// TIA Portal V15.1 export
// export: Created 2020-06-12T07:35:55.4130859Z, ExportSetting None, DisplayName Totally Integrated Automation Portal, DisplayVersion V15.1, DisplayName TIA Portal Openness, DisplayVersion V15.1, DisplayName STEP 7 Professional, DisplayVersion V15.1, DisplayName STEP 7 Safety, DisplayVersion V15.1, DisplayName WinCC Advanced, DisplayVersion V15.1
FUNCTION "SLAG_ctrl" : Void   // FC120, FBD
TITLE = Slag addition base control
{ S7_Optimized_Access := 'TRUE' }
// stored: SetENOAutomatically False
   VAR_TEMP
      tReqFeedOn : Bool;
      tReqFeedOff : Bool;
      tReqPush : Bool;
      tReqDummy : Bool;
      tReqFloodOn : Bool;
      tReqFloodOff : Bool;
      tReqMan : Bool;
      tReqAuto : Bool;
      tReqSetTara : Bool;
      tReqCondMode : Bool;
      tReqDirectMode : Bool;
      tReqRateFree : Bool;
      tReqRateFixed : Bool;
      tStage : Word;
      tDeskActive : Bool;
      tDeskFeedOn : Bool;
      tDeskPush : Bool;
      tManCmdOn : Bool;
      tManCmdOff : Bool;
      tLock : Bool;
      tCmdOn : Bool;
      tCmdOff : Bool;
      tReqOn : Bool;
      tReqOff : Bool;
      tCondStop : Bool;
      tTargetWeightReached : Bool;
      tLoadedWeight : Real;
      tLoadStarting : Bool;
      tLoadStopping : Bool;
      tReqReset : Bool;
      tLock2 : Bool;
      tReqFixSpd2 : Bool;
      tReqFixSpd1 : Bool;
      tInvalidWeight : Bool;
      tNoisedWgt : Real;
      tNoise : Real;
      tDeskChangeSpd : Bool;
      tDeskSelSpd2 : Bool;
      tPwrOk : Bool;
      tDeskSelSpd1 : Bool;
      tDeskFloodOn : Bool;
      tDeskFloodOff : Bool;
      tRestWeight : Real;
      tFeederIsStopped : Bool;
      tBinISEmpty : Bool;
      tHammerBitFast : Bool;
      tHammerBitSlow : Bool;
      tBeat : Bool;
      tLoadRate : Real;
      tReqFloodOff_ : Bool;
   END_VAR
   VAR_TEMP   // added for the SCL form of the ladder/FBD networks
      _w1 : Bool;
      _w2 : Bool;
   END_VAR
BEGIN

REGION Network 1: Common fault
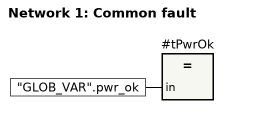
   #tPwrOk := "GLOB_VAR".pwr_ok;
END_REGION

REGION Network 2: HMI request treat
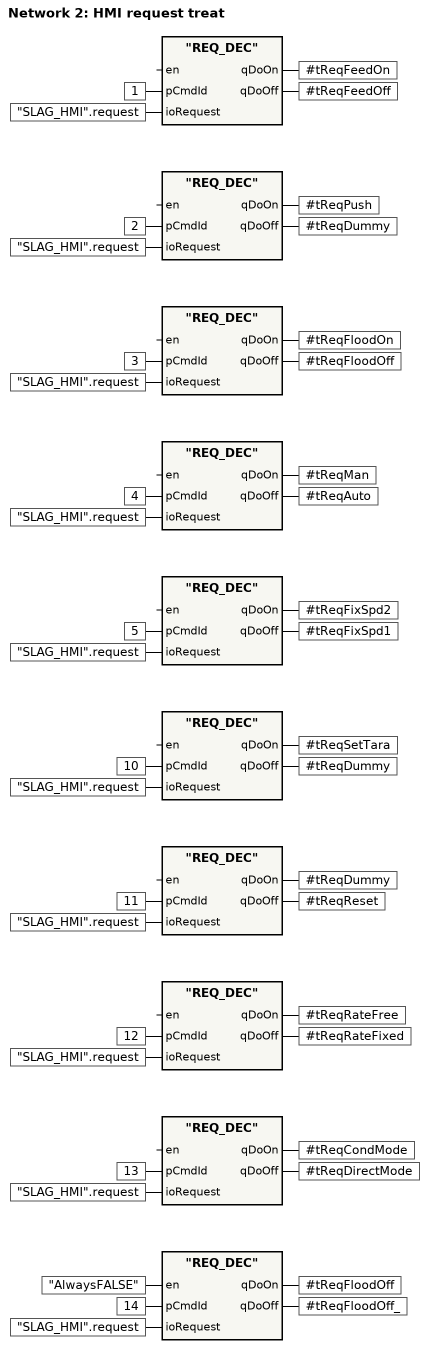
   "REQ_DEC"(pCmdId := 1, ioRequest := "SLAG_HMI".request, qDoOn => #tReqFeedOn, qDoOff => #tReqFeedOff);
   "REQ_DEC"(pCmdId := 2, ioRequest := "SLAG_HMI".request, qDoOn => #tReqPush, qDoOff => #tReqDummy);
   "REQ_DEC"(pCmdId := 3, ioRequest := "SLAG_HMI".request, qDoOn => #tReqFloodOn, qDoOff => #tReqFloodOff);
   "REQ_DEC"(pCmdId := 4, ioRequest := "SLAG_HMI".request, qDoOn => #tReqMan, qDoOff => #tReqAuto);
   "REQ_DEC"(pCmdId := 5, ioRequest := "SLAG_HMI".request, qDoOn => #tReqFixSpd2, qDoOff => #tReqFixSpd1);
   "REQ_DEC"(pCmdId := 10, ioRequest := "SLAG_HMI".request, qDoOn => #tReqSetTara, qDoOff => #tReqDummy);
   "REQ_DEC"(pCmdId := 11, ioRequest := "SLAG_HMI".request, qDoOn => #tReqDummy, qDoOff => #tReqReset);
   "REQ_DEC"(pCmdId := 12, ioRequest := "SLAG_HMI".request, qDoOn => #tReqRateFree, qDoOff => #tReqRateFixed);
   "REQ_DEC"(pCmdId := 13, ioRequest := "SLAG_HMI".request, qDoOn => #tReqCondMode, qDoOff => #tReqDirectMode);
   IF "AlwaysFALSE" THEN
       "REQ_DEC"(pCmdId := 14, ioRequest := "SLAG_HMI".request, qDoOn => #tReqFloodOff, qDoOff => #tReqFloodOff_);
   END_IF;
END_REGION

REGION Network 3: An operators desks are active
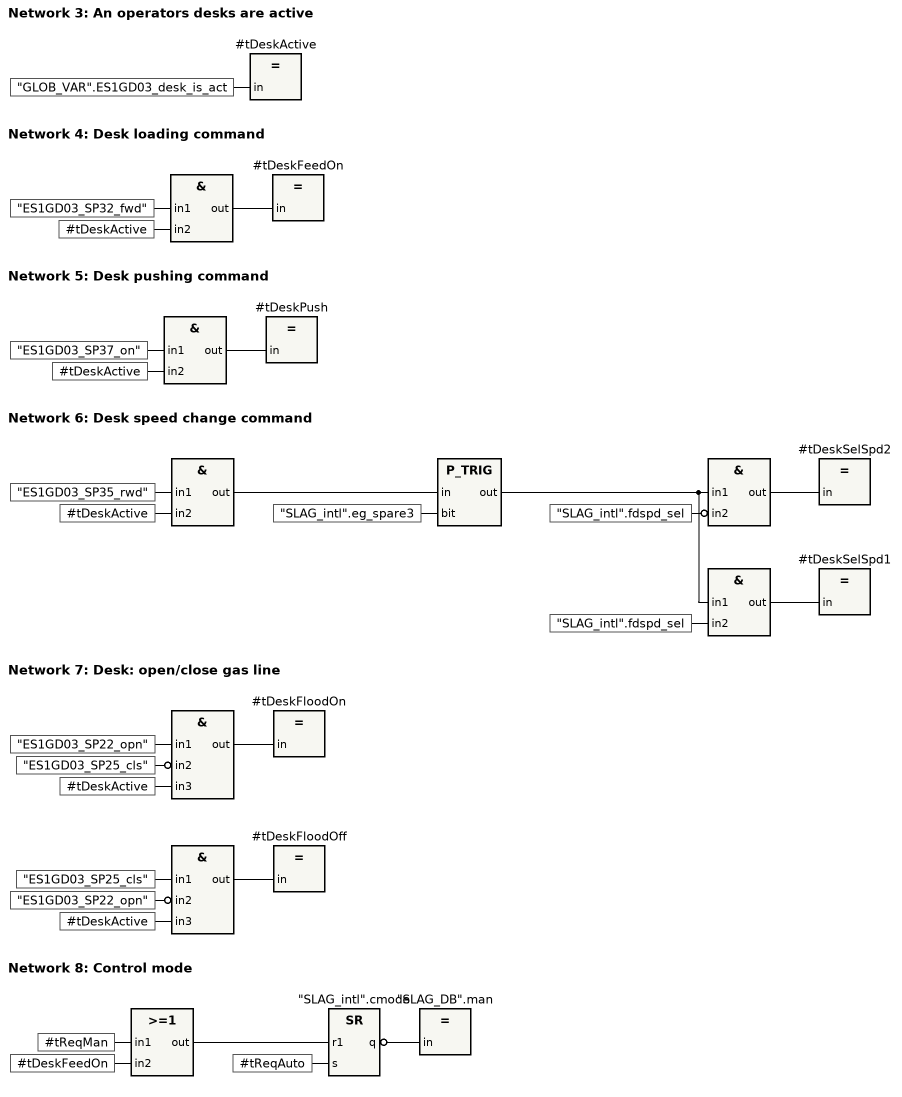
   #tDeskActive := "GLOB_VAR".ES1GD03_desk_is_act;
END_REGION

REGION Network 4: Desk loading command
   #tDeskFeedOn := "ES1GD03_SP32_fwd" AND #tDeskActive;
END_REGION

REGION Network 5: Desk pushing command
   // The sense of this command for a vibro-feeder is not so clear...
   // 
   // But we can use this button to activate the pusher.
   #tDeskPush := "ES1GD03_SP37_on" AND #tDeskActive;
END_REGION

REGION Network 6: Desk speed change command
   #_w1 := "ES1GD03_SP35_rwd" AND #tDeskActive;
   #_w2 := #_w1 AND NOT "SLAG_intl".eg_spare3;   // rising edge
   "SLAG_intl".eg_spare3 := #_w1;
   #tDeskSelSpd2 := #_w2 AND NOT "SLAG_intl".fdspd_sel;
   #tDeskSelSpd1 := #_w2 AND "SLAG_intl".fdspd_sel;
END_REGION

REGION Network 7: Desk: open/close gas line
   #tDeskFloodOn := "ES1GD03_SP22_opn" AND NOT "ES1GD03_SP25_cls" AND #tDeskActive;
   #tDeskFloodOff := "ES1GD03_SP25_cls" AND NOT "ES1GD03_SP22_opn" AND #tDeskActive;
END_REGION

REGION Network 8: Control mode
   // "SLAG_intl".cmode
   IF #tReqAuto THEN
       "SLAG_intl".cmode := TRUE;   // SR flip-flop
   END_IF;
   IF #tReqMan OR #tDeskFeedOn THEN "SLAG_intl".cmode := FALSE; END_IF;
   "SLAG_DB".man := NOT "SLAG_intl".cmode;
END_REGION

REGION Network 9: Loading mode
   // For an external program the conditional loading is always using
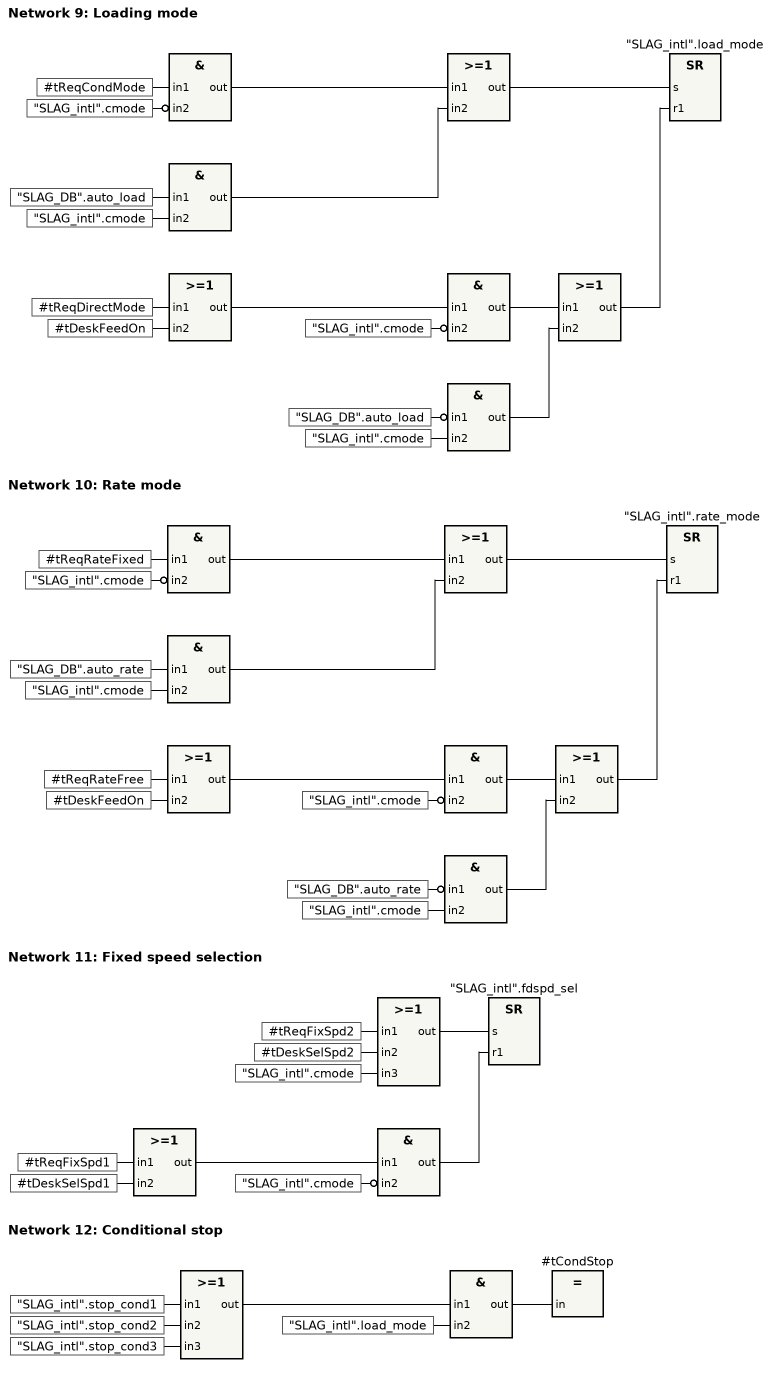
   IF (#tReqCondMode AND NOT "SLAG_intl".cmode) OR ("SLAG_DB".auto_load AND "SLAG_intl".cmode) THEN
       "SLAG_intl".load_mode := TRUE;   // SR flip-flop
   END_IF;
   IF ((#tReqDirectMode OR #tDeskFeedOn) AND NOT "SLAG_intl".cmode) OR (NOT "SLAG_DB".auto_load AND "SLAG_intl".cmode) THEN
       "SLAG_intl".load_mode := FALSE;
   END_IF;
END_REGION

REGION Network 10: Rate mode
   IF (#tReqRateFixed AND NOT "SLAG_intl".cmode) OR ("SLAG_DB".auto_rate AND "SLAG_intl".cmode) THEN
       "SLAG_intl".rate_mode := TRUE;   // SR flip-flop
   END_IF;
   IF ((#tReqRateFree OR #tDeskFeedOn) AND NOT "SLAG_intl".cmode) OR (NOT "SLAG_DB".auto_rate AND "SLAG_intl".cmode) THEN
       "SLAG_intl".rate_mode := FALSE;
   END_IF;
END_REGION

REGION Network 11: Fixed speed selection
   IF #tReqFixSpd2 OR #tDeskSelSpd2 OR "SLAG_intl".cmode THEN
       "SLAG_intl".fdspd_sel := TRUE;   // SR flip-flop
   END_IF;
   IF (#tReqFixSpd1 OR #tDeskSelSpd1) AND NOT "SLAG_intl".cmode THEN "SLAG_intl".fdspd_sel := FALSE; END_IF;
END_REGION

REGION Network 12: Conditional stop
   // NB: This network here becuase of optimization
   #tCondStop := ("SLAG_intl".stop_cond1 OR "SLAG_intl".stop_cond2 OR "SLAG_intl".stop_cond3) AND "SLAG_intl".load_mode;
END_REGION

REGION Network 13: Lock by invalid measurement
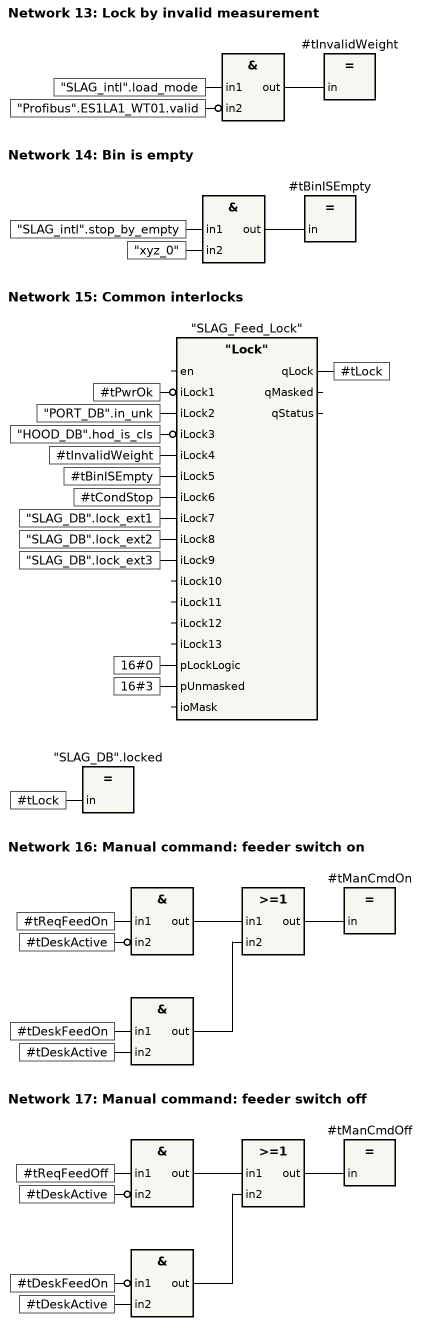
   #tInvalidWeight := "SLAG_intl".load_mode AND NOT "Profibus".ES1LA1_WT01.valid;
END_REGION

REGION Network 14: Bin is empty
   #tBinISEmpty := "SLAG_intl".stop_by_empty AND "xyz_0";
END_REGION

REGION Network 15: Common interlocks
   "SLAG_Feed_Lock"(iLock1 := NOT #tPwrOk,   // "Lock"
                    iLock2 := "PORT_DB".in_unk,
                    iLock3 := NOT "HOOD_DB".hod_is_cls,
                    iLock4 := #tInvalidWeight,
                    iLock5 := #tBinISEmpty,
                    iLock6 := #tCondStop,
                    iLock7 := "SLAG_DB".lock_ext1,
                    iLock8 := "SLAG_DB".lock_ext2,
                    iLock9 := "SLAG_DB".lock_ext3,
                    pLockLogic := 16#0,
                    pUnmasked := 16#3,
                    qLock => #tLock);
   "SLAG_DB".locked := #tLock;
END_REGION

REGION Network 16: Manual command: feeder switch on
   #tManCmdOn := (#tReqFeedOn AND NOT #tDeskActive) OR (#tDeskFeedOn AND #tDeskActive);
END_REGION

REGION Network 17: Manual command: feeder switch off
   #tManCmdOff := (#tReqFeedOff AND NOT #tDeskActive) OR (NOT #tDeskFeedOn AND #tDeskActive);
END_REGION

REGION Network 18: Manual start/stop
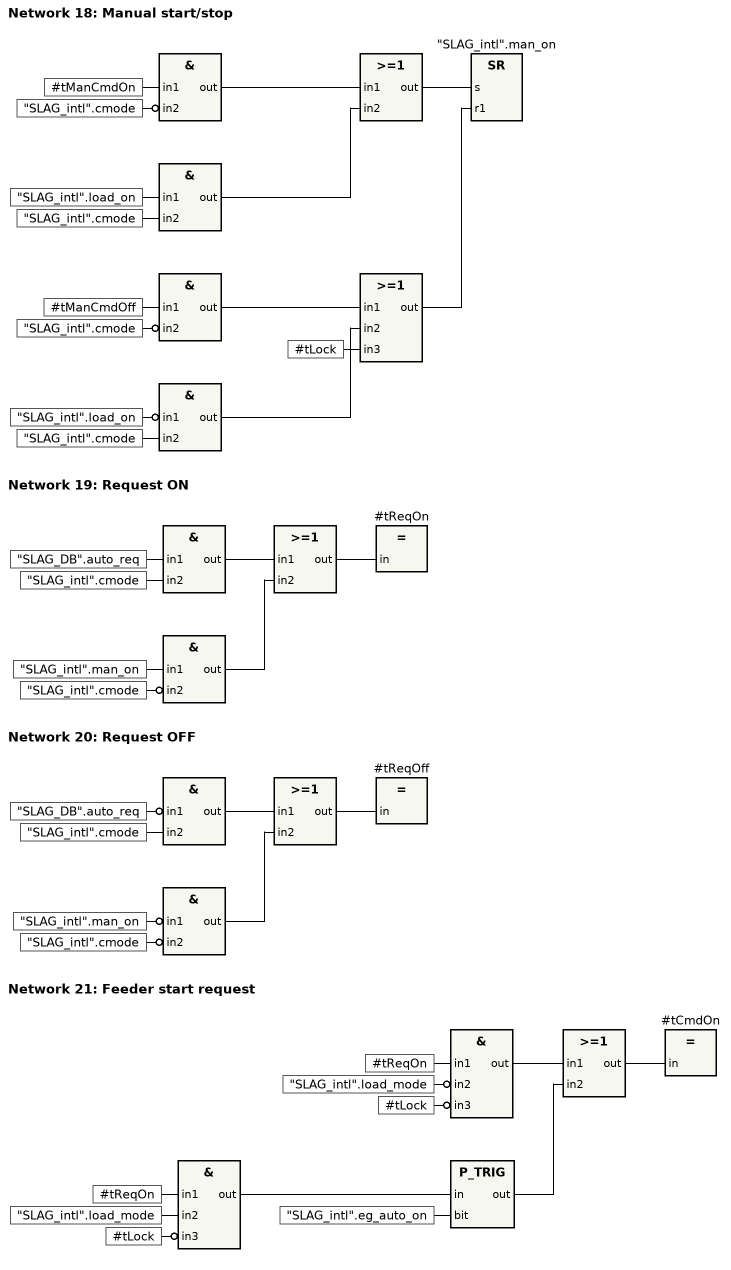
   IF (#tManCmdOn AND NOT "SLAG_intl".cmode) OR ("SLAG_intl".load_on AND "SLAG_intl".cmode) THEN
       "SLAG_intl".man_on := TRUE;   // SR flip-flop
   END_IF;
   IF (#tManCmdOff AND NOT "SLAG_intl".cmode) OR (NOT "SLAG_intl".load_on AND "SLAG_intl".cmode) OR #tLock THEN
       "SLAG_intl".man_on := FALSE;
   END_IF;
END_REGION

REGION Network 19: Request ON
   #tReqOn := ("SLAG_DB".auto_req AND "SLAG_intl".cmode) OR ("SLAG_intl".man_on AND NOT "SLAG_intl".cmode);
END_REGION

REGION Network 20: Request OFF
   #tReqOff := (NOT "SLAG_DB".auto_req AND "SLAG_intl".cmode) OR (NOT "SLAG_intl".man_on AND NOT "SLAG_intl".cmode);
END_REGION

REGION Network 21: Feeder start request
   // I use tLock because want to implmement a restartable program
   #_w1 := #tReqOn AND "SLAG_intl".load_mode AND NOT #tLock;
   #_w2 := #_w1 AND NOT "SLAG_intl".eg_auto_on;   // rising edge
   "SLAG_intl".eg_auto_on := #_w1;
   #tCmdOn := (#tReqOn AND NOT "SLAG_intl".load_mode AND NOT #tLock) OR #_w2;
END_REGION

REGION Network 22: Feeder stop request
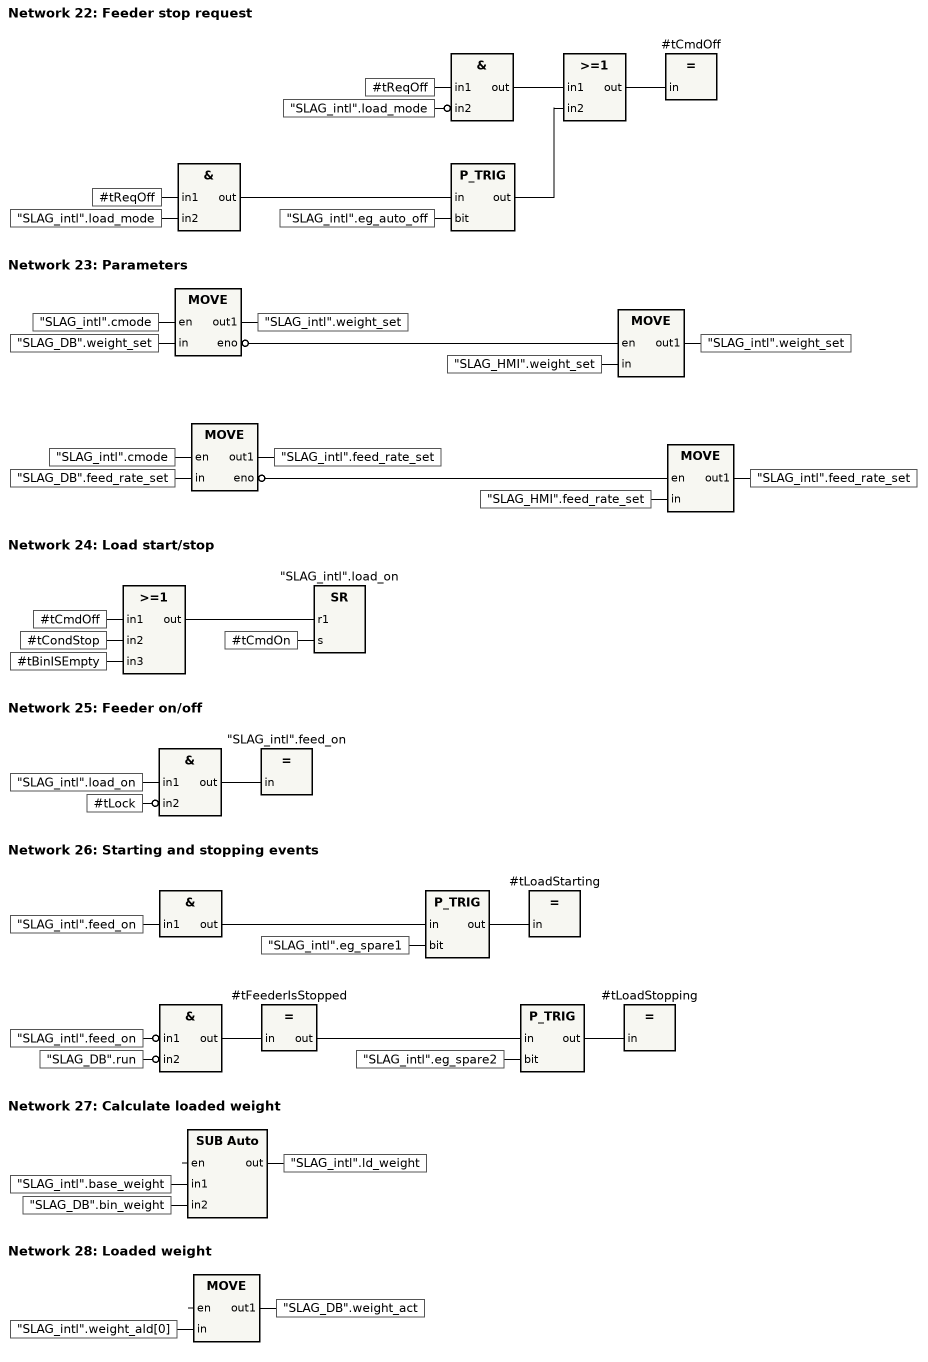
   #_w1 := #tReqOff AND "SLAG_intl".load_mode;
   #_w2 := #_w1 AND NOT "SLAG_intl".eg_auto_off;   // rising edge
   "SLAG_intl".eg_auto_off := #_w1;
   #tCmdOff := (#tReqOff AND NOT "SLAG_intl".load_mode) OR #_w2;
END_REGION

REGION Network 23: Parameters
   IF "SLAG_intl".cmode THEN "SLAG_intl".weight_set := "SLAG_DB".weight_set; END_IF;
   IF NOT "SLAG_intl".cmode THEN "SLAG_intl".weight_set := "SLAG_HMI".weight_set; END_IF;
   IF "SLAG_intl".cmode THEN "SLAG_intl".feed_rate_set := "SLAG_DB".feed_rate_set; END_IF;
   IF NOT "SLAG_intl".cmode THEN "SLAG_intl".feed_rate_set := "SLAG_HMI".feed_rate_set; END_IF;
END_REGION

REGION Network 24: Load start/stop
   IF #tCmdOn THEN
       "SLAG_intl".load_on := TRUE;   // SR flip-flop
   END_IF;
   IF #tCmdOff OR #tCondStop OR #tBinISEmpty THEN "SLAG_intl".load_on := FALSE; END_IF;
END_REGION

REGION Network 25: Feeder on/off
   "SLAG_intl".feed_on := "SLAG_intl".load_on AND NOT #tLock;
END_REGION

REGION Network 26: Starting and stopping events
   #_w1 := "SLAG_intl".feed_on AND NOT "SLAG_intl".eg_spare1;   // rising edge
   "SLAG_intl".eg_spare1 := "SLAG_intl".feed_on;
   #tLoadStarting := #_w1;
   #tFeederIsStopped := NOT "SLAG_intl".feed_on AND NOT "SLAG_DB".run;
   #_w2 := #tFeederIsStopped AND NOT "SLAG_intl".eg_spare2;   // rising edge
   "SLAG_intl".eg_spare2 := #tFeederIsStopped;
   #tLoadStopping := #_w2;
END_REGION

REGION Network 27: Calculate loaded weight
   "SLAG_intl".ld_weight := "SLAG_intl".base_weight - "SLAG_DB".bin_weight;
END_REGION

REGION Network 28: Loaded weight
   "SLAG_DB".weight_act := "SLAG_intl".weight_ald[0];
END_REGION

REGION Network 29: Calculate accumulating loaded weight
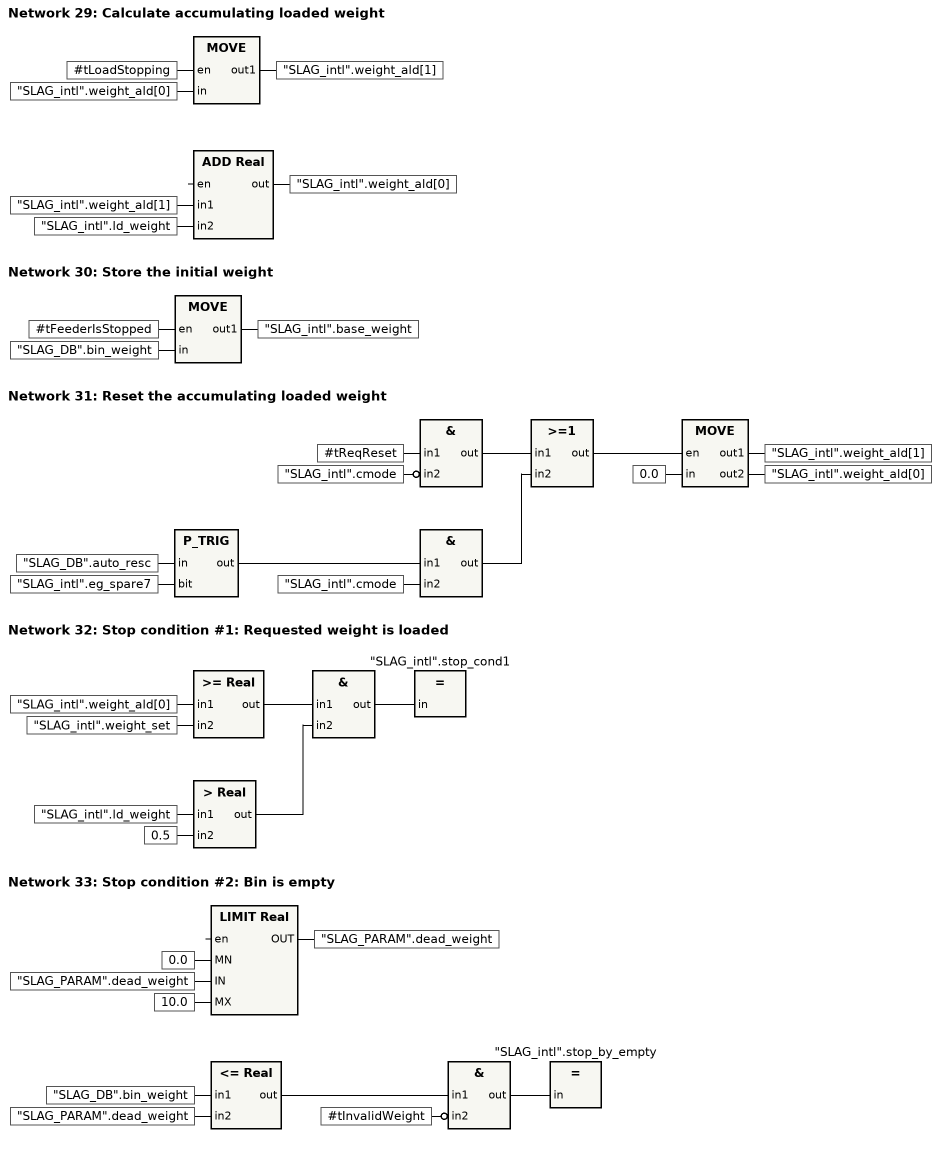
   IF #tLoadStopping THEN "SLAG_intl".weight_ald[1] := "SLAG_intl".weight_ald[0]; END_IF;
   "SLAG_intl".weight_ald[0] := "SLAG_intl".weight_ald[1] + "SLAG_intl".ld_weight;
END_REGION

REGION Network 30: Store the initial weight
   // The #tLoadStarting has been replace by {NOT "SLAG_intl".feed_on }
   IF #tFeederIsStopped THEN "SLAG_intl".base_weight := "SLAG_DB".bin_weight; END_IF;
END_REGION

REGION Network 31: Reset the accumulating loaded weight
   #_w1 := "SLAG_DB".auto_resc AND NOT "SLAG_intl".eg_spare7;   // rising edge
   "SLAG_intl".eg_spare7 := "SLAG_DB".auto_resc;
   IF (#tReqReset AND NOT "SLAG_intl".cmode) OR (#_w1 AND "SLAG_intl".cmode) THEN
       "SLAG_intl".weight_ald[1] := 0.0;
       "SLAG_intl".weight_ald[0] := 0.0;
   END_IF;
END_REGION

REGION Network 32: Stop condition #1: Requested weight is loaded
   "SLAG_intl".stop_cond1 := ("SLAG_intl".weight_ald[0] >= "SLAG_intl".weight_set) AND ("SLAG_intl".ld_weight > 0.5);
END_REGION

REGION Network 33: Stop condition #2: Bin is empty
   "SLAG_PARAM".dead_weight := LIMIT(MN := 0.0, IN := "SLAG_PARAM".dead_weight, MX := 10.0);
   "SLAG_intl".stop_by_empty := ("SLAG_DB".bin_weight <= "SLAG_PARAM".dead_weight) AND NOT #tInvalidWeight;
END_REGION

REGION Network 34: Detect a prestop weight
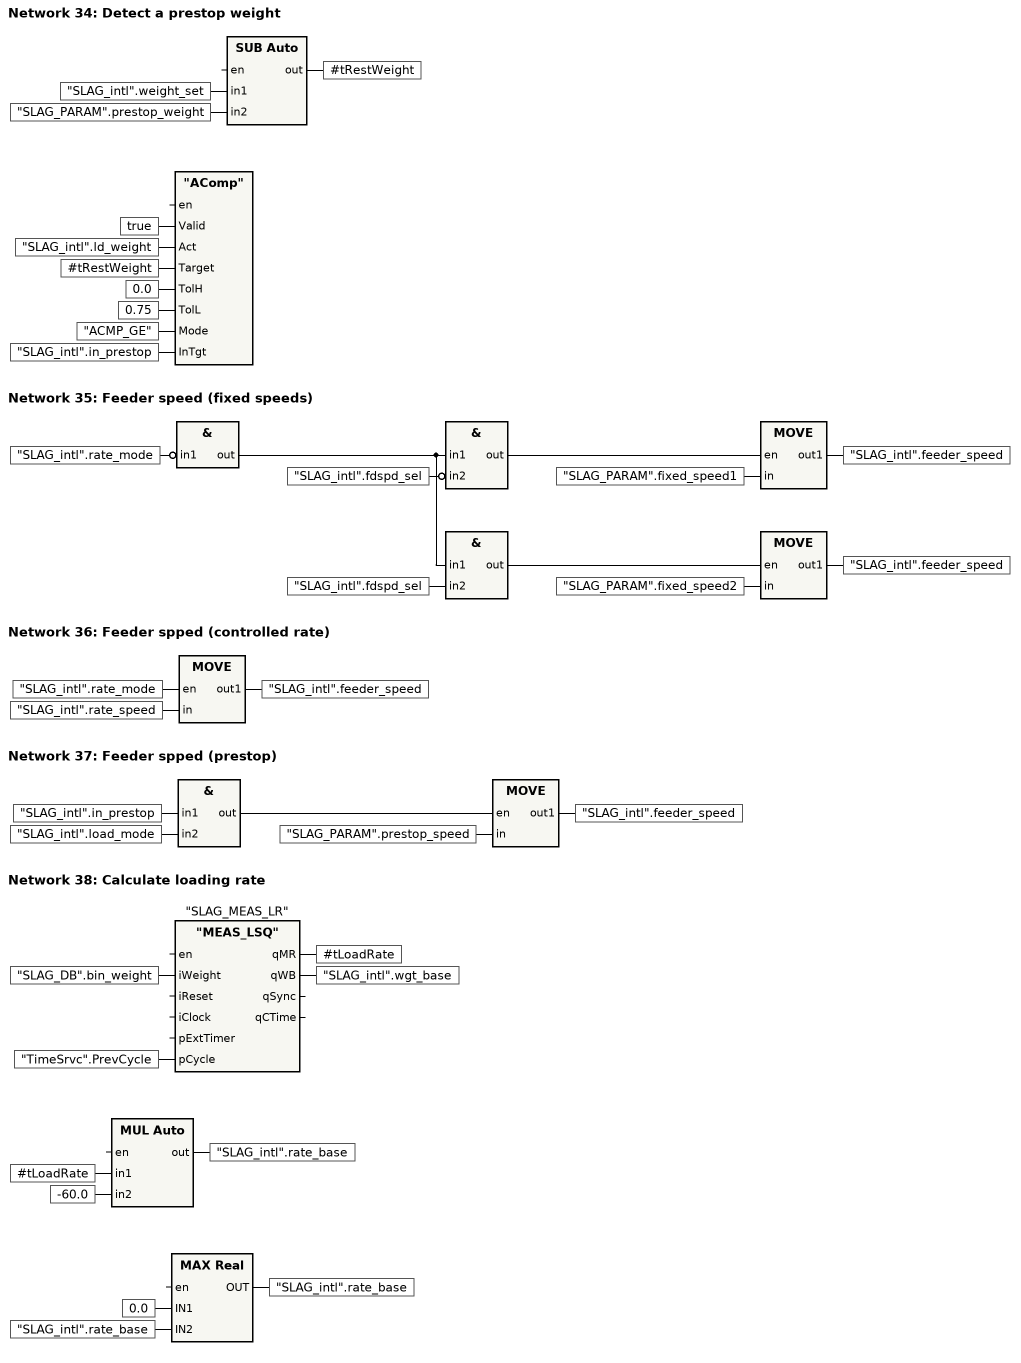
   #tRestWeight := "SLAG_intl".weight_set - "SLAG_PARAM".prestop_weight;
   "AComp"(Valid := true,
           Act := "SLAG_intl".ld_weight,
           Target := #tRestWeight,
           TolH := 0.0,
           TolL := 0.75,
           Mode := "ACMP_GE",
           InTgt := "SLAG_intl".in_prestop);
END_REGION

REGION Network 35: Feeder speed (fixed speeds)
   #_w1 := NOT "SLAG_intl".rate_mode;
   IF #_w1 AND NOT "SLAG_intl".fdspd_sel THEN "SLAG_intl".feeder_speed := "SLAG_PARAM".fixed_speed1; END_IF;
   IF #_w1 AND "SLAG_intl".fdspd_sel THEN "SLAG_intl".feeder_speed := "SLAG_PARAM".fixed_speed2; END_IF;
END_REGION

REGION Network 36: Feeder spped (controlled rate)
   IF "SLAG_intl".rate_mode THEN "SLAG_intl".feeder_speed := "SLAG_intl".rate_speed; END_IF;
END_REGION

REGION Network 37: Feeder spped (prestop)
   IF "SLAG_intl".in_prestop AND "SLAG_intl".load_mode THEN
       "SLAG_intl".feeder_speed := "SLAG_PARAM".prestop_speed;
   END_IF;
END_REGION

REGION Network 38: Calculate loading rate
   "SLAG_MEAS_LR"(iWeight := "SLAG_DB".bin_weight,   // "MEAS_LSQ"
                  pCycle := "TimeSrvc".PrevCycle,
                  qMR => #tLoadRate,
                  qWB => "SLAG_intl".wgt_base);
   "SLAG_intl".rate_base := #tLoadRate * (-60.0);
   "SLAG_intl".rate_base := MAX(IN1 := 0.0, IN2 := "SLAG_intl".rate_base);
END_REGION

REGION Network 39: Stacking detection
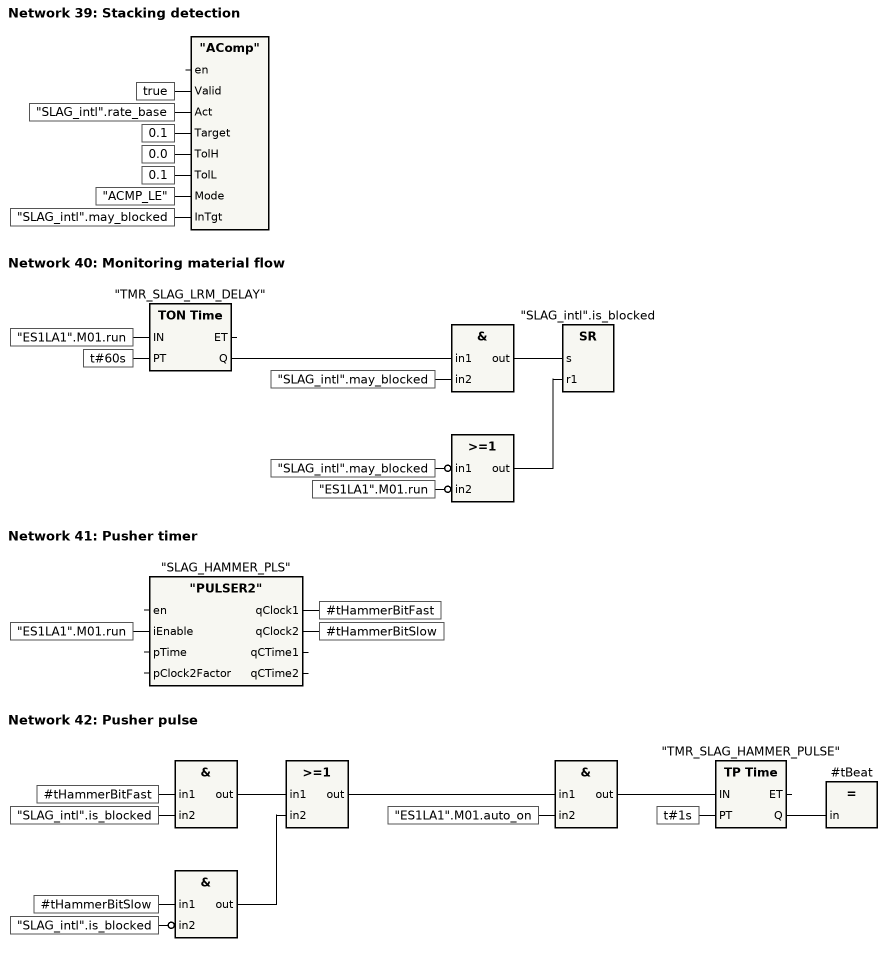
   "AComp"(Valid := true,
           Act := "SLAG_intl".rate_base,
           Target := 0.1,
           TolH := 0.0,
           TolL := 0.1,
           Mode := "ACMP_LE",
           InTgt := "SLAG_intl".may_blocked);
END_REGION

REGION Network 40: Monitoring material flow
   "TMR_SLAG_LRM_DELAY".TON(IN := "ES1LA1".M01.run, PT := t#60s);
   IF "TMR_SLAG_LRM_DELAY".Q AND "SLAG_intl".may_blocked THEN
       "SLAG_intl".is_blocked := TRUE;   // SR flip-flop
   END_IF;
   IF NOT "SLAG_intl".may_blocked OR NOT "ES1LA1".M01.run THEN "SLAG_intl".is_blocked := FALSE; END_IF;
END_REGION

REGION Network 41: Pusher timer
   "SLAG_HAMMER_PLS"(iEnable := "ES1LA1".M01.run, qClock1 => #tHammerBitFast, qClock2 => #tHammerBitSlow);   // "PULSER2"
END_REGION

REGION Network 42: Pusher pulse
   "TMR_SLAG_HAMMER_PULSE".TP(IN := ((#tHammerBitFast AND "SLAG_intl".is_blocked) OR (#tHammerBitSlow AND NOT "SLAG_intl".is_blocked)) AND "ES1LA1".M01.auto_on,
                           PT := t#1s);
   #tBeat := "TMR_SLAG_HAMMER_PULSE".Q;
END_REGION

REGION Network 43: Gas flooding
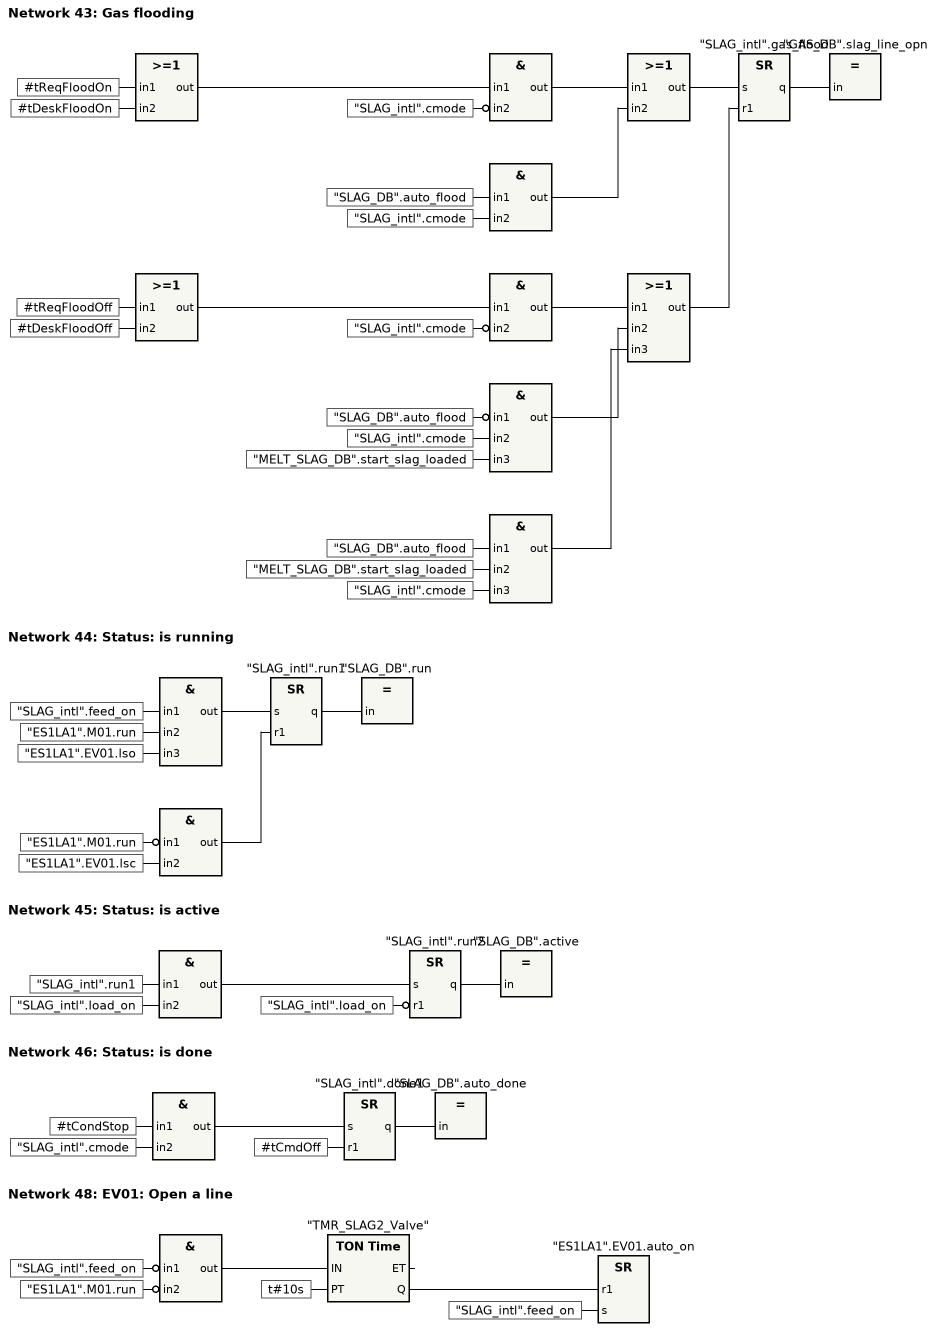
   IF ((#tReqFloodOn OR #tDeskFloodOn) AND NOT "SLAG_intl".cmode) OR ("SLAG_DB".auto_flood AND "SLAG_intl".cmode) THEN
       "SLAG_intl".gas_flood := TRUE;   // SR flip-flop
   END_IF;
   IF ((#tReqFloodOff OR #tDeskFloodOff) AND NOT "SLAG_intl".cmode) OR (NOT "SLAG_DB".auto_flood AND "SLAG_intl".cmode AND "MELT_SLAG_DB".start_slag_loaded) OR ("SLAG_DB".auto_flood AND "MELT_SLAG_DB".start_slag_loaded AND "SLAG_intl".cmode) THEN
       "SLAG_intl".gas_flood := FALSE;
   END_IF;
   "GAS_DB".slag_line_opn := "SLAG_intl".gas_flood;
END_REGION

REGION Network 44: Status: is running
   IF "SLAG_intl".feed_on AND "ES1LA1".M01.run AND "ES1LA1".EV01.lso THEN
       "SLAG_intl".run1 := TRUE;   // SR flip-flop
   END_IF;
   IF NOT "ES1LA1".M01.run AND "ES1LA1".EV01.lsc THEN "SLAG_intl".run1 := FALSE; END_IF;
   "SLAG_DB".run := "SLAG_intl".run1;
END_REGION

REGION Network 45: Status: is active
   IF "SLAG_intl".run1 AND "SLAG_intl".load_on THEN
       "SLAG_intl".run2 := TRUE;   // SR flip-flop
   END_IF;
   IF NOT "SLAG_intl".load_on THEN "SLAG_intl".run2 := FALSE; END_IF;
   "SLAG_DB".active := "SLAG_intl".run2;
END_REGION

REGION Network 46: Status: is done
   IF #tCondStop AND "SLAG_intl".cmode THEN
       "SLAG_intl".done1 := TRUE;   // SR flip-flop
   END_IF;
   IF #tCmdOff THEN "SLAG_intl".done1 := FALSE; END_IF;
   "SLAG_DB".auto_done := "SLAG_intl".done1;
END_REGION

REGION Network 47: [ DEVICES control]
END_REGION

REGION Network 48: EV01: Open a line
   "TMR_SLAG2_Valve".TON(IN := NOT "SLAG_intl".feed_on AND NOT "ES1LA1".M01.run, PT := t#10s);
   IF "SLAG_intl".feed_on THEN
       "ES1LA1".EV01.auto_on := TRUE;   // SR flip-flop
   END_IF;
   IF "TMR_SLAG2_Valve".Q THEN "ES1LA1".EV01.auto_on := FALSE; END_IF;
END_REGION

REGION Network 49: EV01: lock open
   // I do not want to use the lock, to avoid a valve closing while a loading
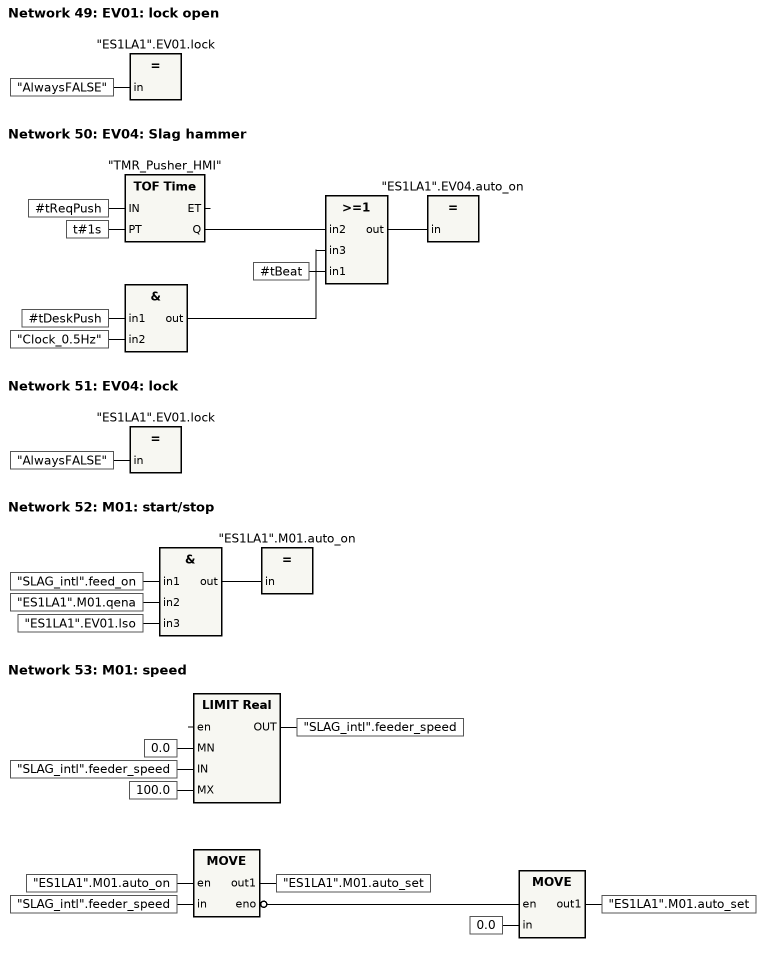
   "ES1LA1".EV01.lock := "AlwaysFALSE";
END_REGION

REGION Network 50: EV04: Slag hammer
   "TMR_Pusher_HMI".TOF(IN := #tReqPush, PT := t#1s);
   "ES1LA1".EV04.auto_on := "TMR_Pusher_HMI".Q OR (#tDeskPush AND "Clock_0.5Hz") OR #tBeat;
END_REGION

REGION Network 51: EV04: lock
   // there are not the restrictions
   "ES1LA1".EV01.lock := "AlwaysFALSE";
END_REGION

REGION Network 52: M01: start/stop
   "ES1LA1".M01.auto_on := "SLAG_intl".feed_on AND "ES1LA1".M01.qena AND "ES1LA1".EV01.lso;
END_REGION

REGION Network 53: M01: speed
   "SLAG_intl".feeder_speed := LIMIT(MN := 0.0, IN := "SLAG_intl".feeder_speed, MX := 100.0);
   IF "ES1LA1".M01.auto_on THEN "ES1LA1".M01.auto_set := "SLAG_intl".feeder_speed; END_IF;
   IF NOT "ES1LA1".M01.auto_on THEN "ES1LA1".M01.auto_set := 0.0; END_IF;
END_REGION

REGION Network 54: M01: lock forward
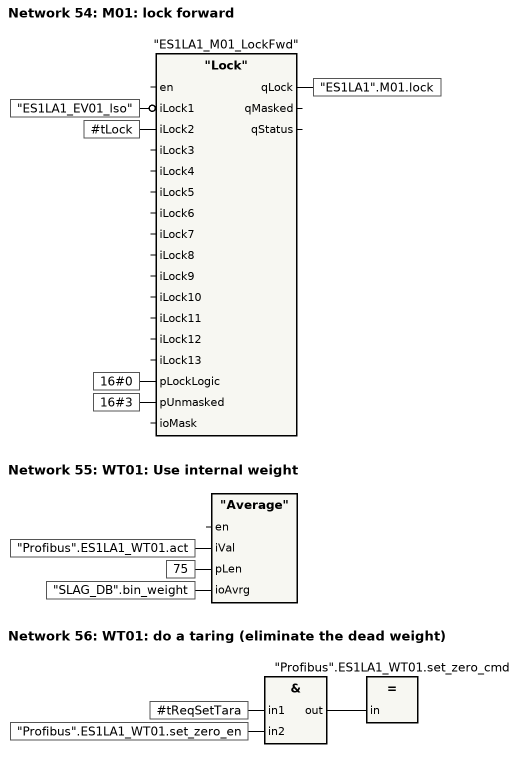
   "ES1LA1_M01_LockFwd"(iLock1 := NOT "ES1LA1_EV01_lso",   // "Lock"
                        iLock2 := #tLock,
                        pLockLogic := 16#0,
                        pUnmasked := 16#3,
                        qLock => "ES1LA1".M01.lock);
END_REGION

REGION Network 55: WT01: Use internal weight
   "Average"(iVal := "Profibus".ES1LA1_WT01.act, pLen := 75, ioAvrg := "SLAG_DB".bin_weight);
END_REGION

REGION Network 56: WT01: do a taring (eliminate the dead weight)
   "Profibus".ES1LA1_WT01.set_zero_cmd := #tReqSetTara AND "Profibus".ES1LA1_WT01.set_zero_en;
END_REGION

REGION Network 57: HMI: status
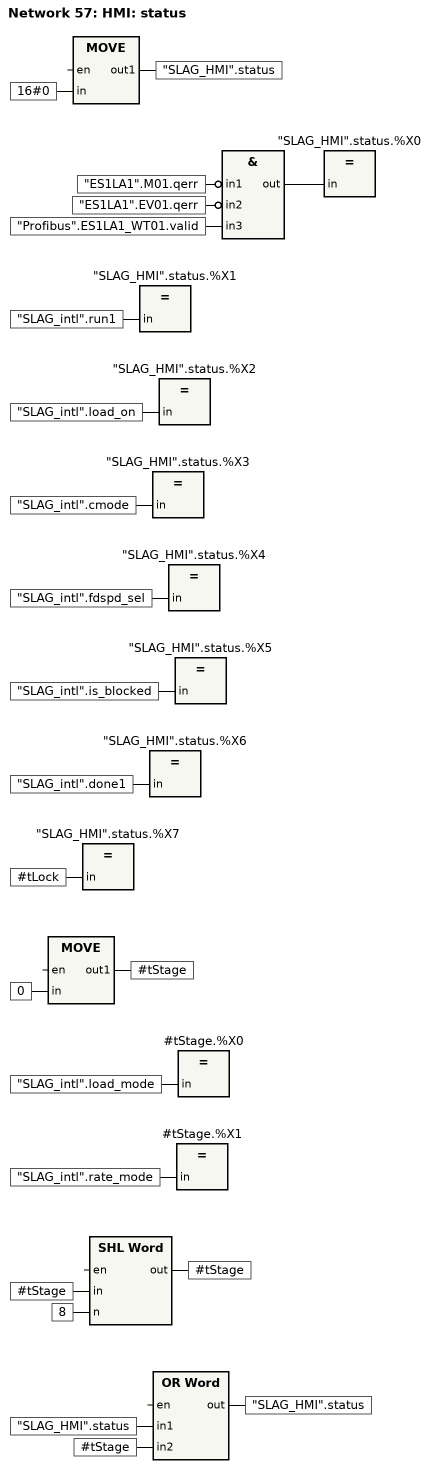
   "SLAG_HMI".status := 16#0;
   "SLAG_HMI".status.%X0 := NOT "ES1LA1".M01.qerr AND NOT "ES1LA1".EV01.qerr AND "Profibus".ES1LA1_WT01.valid;
   "SLAG_HMI".status.%X1 := "SLAG_intl".run1;
   "SLAG_HMI".status.%X2 := "SLAG_intl".load_on;
   "SLAG_HMI".status.%X3 := "SLAG_intl".cmode;
   "SLAG_HMI".status.%X4 := "SLAG_intl".fdspd_sel;
   "SLAG_HMI".status.%X5 := "SLAG_intl".is_blocked;
   "SLAG_HMI".status.%X6 := "SLAG_intl".done1;
   "SLAG_HMI".status.%X7 := #tLock;
   #tStage := 0;
   #tStage.%X0 := "SLAG_intl".load_mode;
   #tStage.%X1 := "SLAG_intl".rate_mode;
   #tStage := SHL(IN := #tStage, N := 8);
   "SLAG_HMI".status := "SLAG_HMI".status OR #tStage;
END_REGION

REGION Network 58: HMI: values
   // This copeing is not sensless :( Not always the physical units have used in a program is good for customer, and visa versa.
   // Yep, this is dummy copeing, but the customer agreed with that units :)
   // And second reson: this method decreases a possibility to damage the important values from HMI
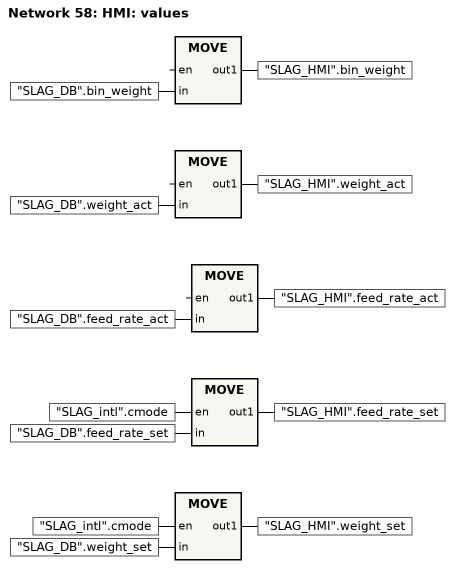
   "SLAG_HMI".bin_weight := "SLAG_DB".bin_weight;
   "SLAG_HMI".weight_act := "SLAG_DB".weight_act;
   "SLAG_HMI".feed_rate_act := "SLAG_DB".feed_rate_act;
   IF "SLAG_intl".cmode THEN
       "SLAG_HMI".feed_rate_set := "SLAG_DB".feed_rate_set;
       "SLAG_HMI".weight_set := "SLAG_DB".weight_set;
   END_IF;
END_REGION
END_FUNCTION
